# EPICS substitutions: db/Festo/ecmcFesto-CMMT-ST_CSP.substitutions
file "ecmcFesto-CMM-ST.template" { pattern
  { CH_ID }
  { 01    }
}

file "ecmcFesto-CMM-ST_Enc.template" { pattern
  { CH_ID }
  { 01    }
  { 02    }
}
